SUBAPPLICATION modbus_tcp (* Subapplication Type *)
  (* Standard: 61499-2 *)
  (* Version 1.0, 2025-01-31, franz *)
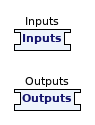
  SUBAPPS
    Outputs : Outputs;
    Inputs : Inputs;
  END_SUBAPPS
END_SUBAPPLICATION
